(* CoDeSys 2.3 export: TDELUTIONSIGNAL.EXP *)

(* Data type *)
TYPE tDelutionSignal : REAL;
END_TYPE
